RESOURCE_TYPE _CBCore1
  (* Standard: 61499-2 *)
  (* Version 0.1, 2019-00-29, hpea485, UOA *)
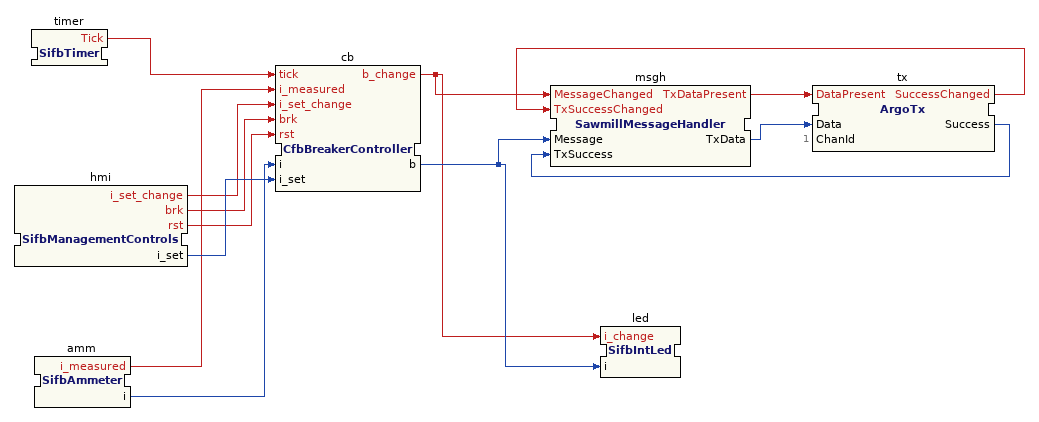
  FBS
    cb : CfbBreakerController;
    msgh : SawmillMessageHandler;
    tx : ArgoTx(ChanId := 1);
    led : SifbIntLed;
    timer : SifbTimer;
    hmi : SifbManagementControls;
    amm : SifbAmmeter;
  END_FBS
  EVENT_CONNECTIONS
    cb.b_change TO msgh.MessageChanged;
    cb.b_change TO led.i_change;
    msgh.TxDataPresent TO tx.DataPresent;
    tx.SuccessChanged TO msgh.TxSuccessChanged;
    timer.Tick TO cb.tick;
    hmi.i_set_change TO cb.i_set_change;
    hmi.brk TO cb.brk;
    hmi.rst TO cb.rst;
    amm.i_measured TO cb.i_measured;
  END_CONNECTIONS
  DATA_CONNECTIONS
    cb.b TO msgh.Message;
    cb.b TO led.i;
    msgh.TxData TO tx.Data;
    tx.Success TO msgh.TxSuccess;
    hmi.i_set TO cb.i_set;
    amm.i TO cb.i;
  END_CONNECTIONS
END_RESOURCE_TYPE
